FUNCTION_BLOCK TwoConveyor (* Composite Function Block Type *)
  (* Standard: 61499-2 *)
  (* Version 0.2, 2003-12-05, JHC, Rockwell Automation, Renamed from NEWCOMPFB. *)
  (* Version 0.1, 2002-01-08, JHC, Rockwell Automation, Added DLY FB as example. *)
  (* Version 0.0, 2000-05-27, JHC, Rockwell Automation *)
  (* Compiler header: package fb.rt.cs725; *)
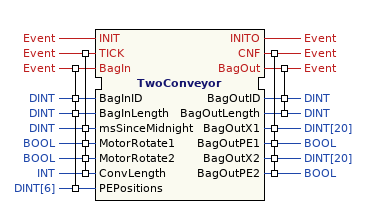
  EVENT_INPUT
    INIT; (* Initialization Request *)
    TICK WITH msSinceMidnight, MotorRotate1, MotorRotate2, ConvLength; (* Normal Execution Request *)
    BagIn WITH BagInID, BagInLength, PEPositions;
  END_EVENT
  EVENT_OUTPUT
    INITO; (* Initialization Confirm *)
    CNF WITH BagOutX1, BagOutPE1, BagOutX2, BagOutPE2; (* Execution Confirmation *)
    BagOut WITH BagOutID, BagOutLength;
  END_EVENT
  VAR_INPUT
    BagInID : DINT;
    BagInLength : DINT;
    msSinceMidnight : DINT;
    MotorRotate1 : BOOL;
    MotorRotate2 : BOOL;
    ConvLength : INT;
    PEPositions : ARRAY [0..5] OF DINT;
  END_VAR
  VAR_OUTPUT
    BagOutID : DINT;
    BagOutLength : DINT;
    BagOutX1 : ARRAY [0..19] OF DINT;
    BagOutPE1 : BOOL;
    BagOutX2 : ARRAY [0..19] OF DINT;
    BagOutPE2 : BOOL;
  END_VAR
  FBS
    C1 : Conveyor_Model_WithNetwork;
    C5 : Conveyor_Model_WithNetwork;
  END_FBS
  EVENT_CONNECTIONS
    TICK TO C1.TICK;
    BagIn TO C1.BagIn;
    C5.CNF TO CNF;
    C5.INITO TO INITO;
    C5.BagOut TO BagOut;
    INIT TO C1.INIT;
    C1.INITO TO C5.INIT;
    C1.CNF TO C5.TICK;
    C1.BagOut TO C5.BagIn;
  END_CONNECTIONS
  DATA_CONNECTIONS
    BagInID TO C1.BagInID;
    BagInLength TO C1.BagInLength;
    msSinceMidnight TO C1.msSinceMidnight;
    MotorRotate1 TO C1.MotorForward;
    C5.BagOutID TO BagOutID;
    C5.BagOutLength TO BagOutLength;
    ConvLength TO C1.ConvLength;
    PEPositions TO C1.PEPositions;
    ConvLength TO C5.ConvLength;
    PEPositions TO C5.PEPositions;
    C1.BagOutPE TO BagOutPE1;
    msSinceMidnight TO C5.msSinceMidnight;
    C1.BagOutX TO BagOutX1;
    C1.BagOutID TO C5.BagInID;
    C1.BagOutLength TO C5.BagInLength;
    MotorRotate2 TO C5.MotorForward;
    C5.BagOutX TO BagOutX2;
    C5.BagOutPE TO BagOutPE2;
  END_CONNECTIONS
END_FUNCTION_BLOCK
